PROGRAM MAIN
VAR
END_VAR

END_PROGRAM

(* stored: Version 1.1.0.1
   POU MAIN: Id {5b0c8ee7-9f57-4395-b71b-9f96424ce740} *)
